(* IEC 61131-3 sources: 2026_Projet_YGO_ExcavatriceDragage/CODE/IO, 4 files *)

(* ---- GVL_IN.st ---- *)
(* ═══════════════════════════════════════════════════════════════
   🗂️ GVL_IN — Entrées machine CONDITIONNÉES (sortie de FB_InputsMachine)
   ───────────────────────────────────────────────────────────────
   📄 Doc : DOC/AF_Partie6_IO_Conditioning_v1.2.md §5
   🔴 ÉCRITURE : FB_InputsMachine SEULEMENT — ne jamais écrire ailleurs !
   ✅ LECTURE : tous les autres POUs (Safety, Winch, Chariot, Homing…)

   🔌 RÈGLE CÂBLAGE SÉCURITÉ (lire avant de modifier) :
   ─────────────────────────────────────────────────────
   Tous les capteurs de sécurité sont câblés en NORMALEMENT FERMÉ (NC) :
     ✅ REPOS / SAIN = TRUE (1) → circuit fermé, courant qui passe → tout va bien
     🔴 DÉFAUT / FIN DE COURSE = FALSE (0) → circuit ouvert (sécurité OU fil coupé)
   Avantage : une coupure de fil = une détection de défaut automatique !
   ═══════════════════════════════════════════════════════════════ *)

// === DECLARATION (à coller dans la partie déclaration du GVL GVL_IN) ===

VAR_GLOBAL

    // ─────────────────────────────────────────────────────────────────────
    // 🛑 SÉCURITÉS COMMUNES (NC — repos = TRUE, défaut/actionné = FALSE)
    // ─────────────────────────────────────────────────────────────────────

    EmergencyStopOk      : BOOL;
    // 🚨 Chaîne arrêt d'urgence (AU bouton champignon + filets de sécurité)
    //    TRUE  = chaîne AU FERMÉE → machine autorisée à bouger
    //    FALSE = chaîne AU COUPÉE (bouton appuyé OU câble coupé) → STOP immédiat

    TopPositionSensor    : BOOL;
    // 🔝 Capteur fin de course HAUT (NC monté en sécurité positive)
    //    TRUE  = capteur LIBRE → câble pas en butée haute, mouvement OK
    //    FALSE = capteur ACTIONNÉ (butée atteinte) → remontée interdite, homing déclenché

    SlackCableSwitch     : BOOL;
    // 🔗 Détecteur mou de câble (NC — repos = câble tendu)
    //    TRUE  = câble TENDU → OK pour descendre
    //    FALSE = câble MOU détecté → descente interdite, remontée autorisée uniquement
    //    ⚠️ Logique de commande : ForbidDescent := NOT SlackCableSwitch (voir FB_Safety_Winch)

    PhaseRotationOk      : BOOL;
    // ⚡ Relais contrôle rotation de phases électriques (NC)
    //    TRUE  = phases CORRECTES → moteurs autorisés à démarrer
    //    FALSE = phases inversées/absentes → SafeStop immédiat (moteurs tourneraient à l'envers !)

    // ─────────────────────────────────────────────────────────────────────
    // 🪝 TREUIL M1 — Retours contacteurs & sécurités (logique mixte NC/NO)
    // ─────────────────────────────────────────────────────────────────────

    M1ContactorFeedbackFwd : BOOL;
    // 📡 Retour contacteur MONTÉE M1 (NO miroir de la bobine)
    //    TRUE  = contacteur montée FERMÉ (bobine alimentée, courant de puissance qui passe)
    //    FALSE = contacteur ouvert (commande coupée ou contacteur collé si commande=TRUE)

    M1ContactorFeedbackRev : BOOL;
    // 📡 Retour contacteur DESCENTE M1 (NO miroir de la bobine)
    //    TRUE  = contacteur descente FERMÉ
    //    FALSE = contacteur ouvert

    M1ThermalFeedback      : BOOL;
    // 🌡️ Sonde thermique moteur M1 (NC — protection moteur contre surchauffe)
    //    TRUE  = température NORMALE → moteur autorisé
    //    FALSE = SURCHAUFFE ou fil coupé → SafeStop M1 immédiat

    M1BrakeFeedback        : BOOL;
    // 🔒 Retour contacteur frein électromagnétique M1 (NC — frein serré = sûr)
    //    TRUE  = frein SERRÉ (bobine coupée, ressort actif) → position sécurisée
    //    FALSE = frein DESSERRÉ (bobine alimentée, frein relâché pour mouvement)

    // ─────────────────────────────────────────────────────────────────────
    // 🪝 TREUIL M2 — Retours contacteurs & sécurités (même logique que M1)
    // ─────────────────────────────────────────────────────────────────────

    M2ContactorFeedbackFwd : BOOL;
    // 📡 Retour contacteur MONTÉE M2 — même logique que M1ContactorFeedbackFwd

    M2ContactorFeedbackRev : BOOL;
    // 📡 Retour contacteur DESCENTE M2 — même logique que M1ContactorFeedbackRev

    M2ThermalFeedback      : BOOL;
    // 🌡️ Sonde thermique moteur M2 — même logique que M1ThermalFeedback

    M2BrakeFeedback        : BOOL;
    // 🔒 Retour contacteur frein M2 — même logique que M1BrakeFeedback

    // ─────────────────────────────────────────────────────────────────────
    // ↔️ CHARIOT M3 — Capteurs de position (NO — actionné = position atteinte = TRUE)
    // ─────────────────────────────────────────────────────────────────────

    ChariotPosFosse1      : BOOL;
    // 📍 Capteur position FOSSE 1 (NO — position atteinte = TRUE)
    //    TRUE  = chariot EN POSITION fosse 1 (fin de course actionné physiquement)
    //    FALSE = chariot hors de la fosse 1

    ChariotPosFosse2      : BOOL;
    // 📍 Capteur position FOSSE 2 — même logique que ChariotPosFosse1

    ChariotPosMaintenance : BOOL;
    // 🔧 Capteur position MAINTENANCE — chariot en position de service
    //    TRUE  = position maintenance atteinte (pour interventions mécaniques)

    ChariotPosTremie      : BOOL;
    // 🗑️ Capteur position TRÉMIE (déversement) — chariot en position vidange
    //    TRUE  = position trémie atteinte → autorisation ouverture grappin

    M3BrakeFeedback       : BOOL;
    // 🔒 Retour contacteur frein chariot M3 — même logique que M1BrakeFeedback

END_VAR

(* ---- GVL_OUT.st ---- *)
(* ═══════════════════════════════════════════════════════════════
   🗂️ GVL_OUT — Commandes déjà rampées des FB métier (entrée de FB_OutputsMachine)
   ───────────────────────────────────────────────────────────────
   📄 Doc métier : DOC/AF_Partie6_IO_Conditioning_v1.2.md §5
   🔧 AJOUT (2026-07-03quindecies, demande utilisateur) : `PRG_MAIN` écrit ICI les
      commandes déjà rampées de `FB_Winch`/`FB_Chariot` par simples affectations
      (naturel en LD : 1 rung = 1 bobine), plutôt que de les passer en paramètres
      d'un appel de FB à 15 entrées (lourd à câbler en Ladder). `FB_OutputsMachine`
      lit ensuite ces variables directement en interne, appelée SANS paramètre.
   ⚠️ Écart assumé à Partie2 §0 ("quasi pas de GVL, sauf échange IHM") — même choix
      pragmatique que `GVL_IN`.
   🔴 Écrit UNIQUEMENT par `PRG_MAIN` (après `FB_Winch`/`FB_Chariot`), lu UNIQUEMENT
      par `FB_OutputsMachine`.
   ═══════════════════════════════════════════════════════════════ *)

// === DECLARATION (à coller dans la partie déclaration du GVL GVL_OUT) ===

VAR_GLOBAL
    // 🪝 WINCH M1
    M1RelayFwd        : BOOL;
    M1RelayRev        : BOOL;
    M1SpeedContactor1 : BOOL;
    M1SpeedContactor2 : BOOL;
    M1SpeedContactor3 : BOOL;
    M1SpeedContactor4 : BOOL;
    M1BrakeCmd        : BOOL;

    // 🪝 WINCH M2
    M2RelayFwd        : BOOL;
    M2RelayRev        : BOOL;
    M2SpeedContactor1 : BOOL;
    M2SpeedContactor2 : BOOL;
    M2SpeedContactor3 : BOOL;
    M2SpeedContactor4 : BOOL;
    M2BrakeCmd        : BOOL;

    // ↔️ CHARIOT M3 — seul BrakeCmd est réel
    ChariotBrakeCmd   : BOOL;
END_VAR

(* ---- FB_InputsMachine.st ---- *)
(* ═══════════════════════════════════════════════════════════════
   📥 FB_InputsMachine — Conditionnement ENTRÉES réelles de toute la machine (1 instance)
   ───────────────────────────────────────────────────────────────
   📄 Doc métier : DOC/AF_Partie6_IO_Conditioning_v1.2.md §5 (historique détaillé : AUDIT
      D52/D60/D61/D64)
   🧭 Interface RÉDUITE (Partie3 §1bis) : compose FB_Input (_COMMON) pour TOUTES les entrées
      TOR réelles (Commun/Winch M1/Winch M2/Chariot M3). Référence DIRECTEMENT les I/O réels
      globales en interne (pas de `*Raw`/`Invert*` câblés depuis `PRG_MAIN`) et écrit ses
      sorties DIRECTEMENT dans `GVL_IN.Xxx` (noms courts, sans suffixe) — appelé SANS
      PARAMÈTRE, rien à récupérer en retour. `InvertLogic`/`ChannelOk` de chaque sous-instance
      restent à leur défaut (FALSE/TRUE) — à FORCER DIRECTEMENT sur la sous-instance en vue
      CODESYS pour inverser NO/NC en mise en service, sans recompiler.
   ℹ️ Note utilisateur : prévu pour être implémenté en LANGAGE LD (Ladder) dans CODESYS pour
      faciliter la maintenance — code ci-dessous = référence ST. `FilterTime` : valeurs
      indicatives (`T#20MS`), à ajuster par voie selon le besoin réel (rebond capteur).
   🔴 NON CÂBLÉS ICI (pas de FB consommateur — FB_Grappin n'existe pas encore) :
      `ConveyorInfeedReady_DI`, `GridDwn_RQ`/`GridUp_RQ`, `HelmetClose_RQ`/`HelmetOpen_RQ`,
      `PosCasque_DI`, `PosGrille_DI`, `ThermHydraulique_DI`.
   ═══════════════════════════════════════════════════════════════ *)

// === DECLARATION (à coller dans la partie déclaration du POU FB_InputsMachine) ===

FUNCTION_BLOCK PUBLIC FB_InputsMachine
VAR
    // 🛑 Commun
    instEmergencyStopOk   : FB_Input;
    instSlackCableSwitch  : FB_Input;
    instTopPositionSensor : FB_Input;
    instCtrlPhaseRotation : FB_Input;   // 🆕 2026-07-03sexdecies — contrôle rotation phases élec.

    // 🪝 Winch M1
    instM1ContactorFwd : FB_Input;
    instM1ContactorRev : FB_Input;
    instM1Thermal      : FB_Input;
    instM1BrakeFeedback: FB_Input;

    // 🪝 Winch M2
    instM2ContactorFwd : FB_Input;
    instM2ContactorRev : FB_Input;
    instM2Thermal      : FB_Input;
    instM2BrakeFeedback: FB_Input;

    // ↔️ Chariot M3
    instChariotPosFosse1      : FB_Input;
    instChariotPosFosse2      : FB_Input;
    instChariotPosMaintenance : FB_Input;
    instChariotPosTremie      : FB_Input;
    instM3BrakeFeedback       : FB_Input;
END_VAR

// === IMPLEMENTATION (à coller dans le corps ST du POU FB_InputsMachine) ===

// 🛑 ─── COMMUN ────────────────────────────────────────────────────────────
// ⚠️ Bypass TEST banc (GVL_DEBUG) — TOUJOURS FALSE avant essai réel avec la chaîne AU câblée
instEmergencyStopOk(InputRaw := EmergencyStopOk_DI OR GVL_DEBUG.DBG_EmergencyStopOkBypass_TEST, FilterTime := T#20MS);
GVL_IN.EmergencyStopOk := instEmergencyStopOk.State;

// ⚠️ Bypass TEST banc (GVL_DEBUG, créé par l'utilisateur) — TOUJOURS FALSE avant essai réel
// avec le vrai capteur mou de câble câblé. Câblage sécurité : TRUE=OK (pas de mou) — le
// bypass force donc l'état OK, cohérent avec les autres bypass (OR sur le signal brut).
instSlackCableSwitch(InputRaw := M1_M2_SlackCableSwitch_DI OR GVL_DEBUG.DBG_SlackCableSwitch_TEST, FilterTime := T#20MS);
GVL_IN.SlackCableSwitch := instSlackCableSwitch.State;

// ⚠️ Bypass TEST banc (GVL_DEBUG) — TOUJOURS FALSE avant essai réel avec le capteur câblé
instTopPositionSensor(InputRaw := M1_M2_TopPositionSensor_DI OR GVL_DEBUG.DBG_TopPositionSensorBypass_TEST, FilterTime := T#20MS);
GVL_IN.TopPositionSensor := instTopPositionSensor.State;

// 🆕 Contrôle rotation phases électriques (2026-07-03sexdecies) — TRUE = rotation correcte.
// Câblé dans FB_Safety_Winch/FB_Safety_Chariot (D71), pas directement sur EmergencyStopOk.
// ⚠️ Bypass TEST banc (GVL_DEBUG, créé par l'utilisateur) — TOUJOURS FALSE avant essai réel
// avec le vrai contrôle de rotation câblé.
instCtrlPhaseRotation(InputRaw := CtrlPhaseRotation_DI OR GVL_DEBUG.DBG_CtrlPhaseRotation_Bypass_TEST, FilterTime := T#20MS);
GVL_IN.PhaseRotationOk := instCtrlPhaseRotation.State;

// 🪝 ─── WINCH M1 ──────────────────────────────────────────────────────────
instM1ContactorFwd(InputRaw := M1_ContactorFeedbackFwd_DI, FilterTime := T#20MS);
GVL_IN.M1ContactorFeedbackFwd := instM1ContactorFwd.State;

instM1ContactorRev(InputRaw := M1_ContactorFeedbackRev_DI, FilterTime := T#20MS);
GVL_IN.M1ContactorFeedbackRev := instM1ContactorRev.State;

instM1Thermal(InputRaw := M1_ThermalFeedback_DI, FilterTime := T#20MS);
GVL_IN.M1ThermalFeedback := instM1Thermal.State;

// 🆕 Retour frein M1 RÉEL (était miroir logiciel GVL_Winch_M1_Stub)
instM1BrakeFeedback(InputRaw := M1_BrakeContactorFeedback_DI, FilterTime := T#20MS);
GVL_IN.M1BrakeFeedback := instM1BrakeFeedback.State;

// 🪝 ─── WINCH M2 ──────────────────────────────────────────────────────────
instM2ContactorFwd(InputRaw := M2_ContactorFeedbackFwd_DI, FilterTime := T#20MS);
GVL_IN.M2ContactorFeedbackFwd := instM2ContactorFwd.State;

instM2ContactorRev(InputRaw := M2_ContactorFeedbackRev_DI, FilterTime := T#20MS);
GVL_IN.M2ContactorFeedbackRev := instM2ContactorRev.State;

instM2Thermal(InputRaw := M2_ThermalFeedback_DI, FilterTime := T#20MS);
GVL_IN.M2ThermalFeedback := instM2Thermal.State;

// 🆕 Retour frein M2 RÉEL (était miroir logiciel GVL_Winch_M2_Stub)
instM2BrakeFeedback(InputRaw := M2_BrakeContactorFeedback_DI, FilterTime := T#20MS);
GVL_IN.M2BrakeFeedback := instM2BrakeFeedback.State;

// ↔️ ─── CHARIOT M3 — 4 capteurs position réels ───────────────────────────
instChariotPosFosse1(InputRaw := PosFosse1_DI, FilterTime := T#20MS);
GVL_IN.ChariotPosFosse1 := instChariotPosFosse1.State;

instChariotPosFosse2(InputRaw := PosFosse2_DI, FilterTime := T#20MS);
GVL_IN.ChariotPosFosse2 := instChariotPosFosse2.State;

instChariotPosMaintenance(InputRaw := PosMaintenance_DI, FilterTime := T#20MS);
GVL_IN.ChariotPosMaintenance := instChariotPosMaintenance.State;

instChariotPosTremie(InputRaw := PosTremie_DI, FilterTime := T#20MS);
GVL_IN.ChariotPosTremie := instChariotPosTremie.State;

// 🆕 Retour frein M3 RÉEL (était miroir logiciel GVL_Chariot_M3_Stub)
instM3BrakeFeedback(InputRaw := M3_BrakeContactorFeedback_DI, FilterTime := T#20MS);
GVL_IN.M3BrakeFeedback := instM3BrakeFeedback.State;

(* ---- PRG_0_Inputs.st ---- *)
(* ═══════════════════════════════════════════════════════════════
   📥 PRG_0_Inputs — Acquisition et conditionnement des ENTRÉES (PROGRAMME)
   ───────────────────────────────────────────────────────────────
   📄 Doc : DOC/AF_Partie6_IO_Conditioning_v1.2.md §5
   ⚙️ Exécuté par la tâche PLC (Task Manager) en position 0.
   ✅ Expose ses sorties en VAR_OUTPUT (lecture seule pour le reste du code).
   ═══════════════════════════════════════════════════════════════ *)

PROGRAM PRG_0_Inputs
VAR_OUTPUT
    // ── 🛑 SÉCURITÉS COMMUNES (NC — repos=TRUE sain, FALSE=défaut/fil coupé) ──────────────
    EmergencyStopOk      : BOOL;   // 🚨 Chaîne AU : TRUE=fermée/armée ✅ | FALSE=AU appuyé ou fil coupé 🔴
    TopPositionSensor    : BOOL;   // 🔝 Fin de course HAUT (NC) : TRUE=libre ✅ | FALSE=butée atteinte 🔴→ForbidAscent
    SlackCableSwitch     : BOOL;   // 🔗 Mou câble sur tambour M2 (NC) : TRUE=câble tendu ✅ | FALSE=mou détecté 🔴→ForbidDescent
    PhaseRotationOk      : BOOL;   // ⚡ Rotation phases élec. (NC) : TRUE=phases OK ✅ | FALSE=inversées/absentes 🔴→SafeStop

    // ── 🪝 TREUIL M1 (contacteurs=NO miroir bobine ; thermique/frein=NC) ────────────────
    M1ContactorFeedbackFwd : BOOL; // 📡 Retour contacteur MONTÉE M1 (NO) : TRUE=contacteur fermé | FALSE=ouvert
    M1ContactorFeedbackRev : BOOL; // 📡 Retour contacteur DESCENTE M1 (NO) : TRUE=contacteur fermé | FALSE=ouvert
    M1ThermalFeedback      : BOOL; // 🌡️ Thermique moteur M1 (NC) : TRUE=temp OK ✅ | FALSE=surchauffe ou coupure 🔴
    M1BrakeFeedback        : BOOL; // 🔒 Retour frein M1 (NC) : TRUE=frein serré repos ✅ | FALSE=desserré/coupure 🔴

    // ── 🪝 TREUIL M2 (même logique que M1) ──────────────────────────────────────────────
    M2ContactorFeedbackFwd : BOOL; // 📡 Retour contacteur MONTÉE M2 (NO) : TRUE=fermé | FALSE=ouvert
    M2ContactorFeedbackRev : BOOL; // 📡 Retour contacteur DESCENTE M2 (NO) : TRUE=fermé | FALSE=ouvert
    M2ThermalFeedback      : BOOL; // 🌡️ Thermique moteur M2 (NC) : TRUE=temp OK ✅ | FALSE=surchauffe ou coupure 🔴
    M2BrakeFeedback        : BOOL; // 🔒 Retour frein M2 (NC) : TRUE=serré repos ✅ | FALSE=desserré/coupure 🔴

    // ── ↔️ CHARIOT M3 (capteurs position=NO — position atteinte=TRUE) ────────────────────
    ChariotPosFosse1      : BOOL;  // 📍 Position fosse 1 (NO) : TRUE=chariot en fosse 1 ✅ | FALSE=absent
    ChariotPosFosse2      : BOOL;  // 📍 Position fosse 2 (NO) : TRUE=chariot en fosse 2 ✅ | FALSE=absent
    ChariotPosMaintenance : BOOL;  // 🔧 Position maintenance (NO) : TRUE=en position service ✅ | FALSE=absent
    ChariotPosTremie      : BOOL;  // 🗑️ Position trémie vidange (NO) : TRUE=en position trémie ✅ | FALSE=absent
    M3BrakeFeedback       : BOOL;  // 🔒 Retour frein chariot M3 (NC) : TRUE=serré repos ✅ | FALSE=desserré 🔴
END_VAR
VAR
    // Instances de filtrage
    instEmergencyStopOk   : FB_Input;
    instSlackCableSwitch  : FB_Input;
    instTopPositionSensor : FB_Input;
    instCtrlPhaseRotation : FB_Input;

    instM1ContactorFwd : FB_Input;
    instM1ContactorRev : FB_Input;
    instM1Thermal      : FB_Input;
    instM1BrakeFeedback: FB_Input;

    instM2ContactorFwd : FB_Input;
    instM2ContactorRev : FB_Input;
    instM2Thermal      : FB_Input;
    instM2BrakeFeedback: FB_Input;

    instChariotPosFosse1      : FB_Input;
    instChariotPosFosse2      : FB_Input;
    instChariotPosMaintenance : FB_Input;
    instChariotPosTremie      : FB_Input;
    instM3BrakeFeedback       : FB_Input;
END_VAR

// === IMPLEMENTATION (corps du PROGRAM PRG_0_Inputs) ===

// 🛑 ─── COMMUN ────────────────────────────────────────────────────────────
instEmergencyStopOk(InputRaw := EmergencyStopOk_DI OR GVL_DEBUG.DBG_EmergencyStopOkBypass_TEST, FilterTime := T#20MS);
EmergencyStopOk := instEmergencyStopOk.State;

instSlackCableSwitch(InputRaw := M1_M2_SlackCableSwitch_DI OR GVL_DEBUG.DBG_SlackCableSwitch_TEST, FilterTime := T#20MS);
SlackCableSwitch := instSlackCableSwitch.State;

instTopPositionSensor(InputRaw := M1_M2_TopPositionSensor_DI OR GVL_DEBUG.DBG_TopPositionSensorBypass_TEST, FilterTime := T#20MS);
TopPositionSensor := instTopPositionSensor.State;

instCtrlPhaseRotation(InputRaw := CtrlPhaseRotation_DI OR GVL_DEBUG.DBG_CtrlPhaseRotation_Bypass_TEST, FilterTime := T#20MS);
PhaseRotationOk := instCtrlPhaseRotation.State;

// 🪝 ─── WINCH M1 ──────────────────────────────────────────────────────────
instM1ContactorFwd(InputRaw := M1_ContactorFeedbackFwd_DI, FilterTime := T#20MS);
M1ContactorFeedbackFwd := instM1ContactorFwd.State;

instM1ContactorRev(InputRaw := M1_ContactorFeedbackRev_DI, FilterTime := T#20MS);
M1ContactorFeedbackRev := instM1ContactorRev.State;

instM1Thermal(InputRaw := M1_ThermalFeedback_DI OR GVL_DEBUG.DBG_ContactorFeedbackBypass_TEST, FilterTime := T#20MS);
M1ThermalFeedback := instM1Thermal.State;

instM1BrakeFeedback(InputRaw := M1_BrakeContactorFeedback_DI, FilterTime := T#20MS);
M1BrakeFeedback := instM1BrakeFeedback.State;

// 🪝 ─── WINCH M2 ──────────────────────────────────────────────────────────
instM2ContactorFwd(InputRaw := M2_ContactorFeedbackFwd_DI, FilterTime := T#20MS);
M2ContactorFeedbackFwd := instM2ContactorFwd.State;

instM2ContactorRev(InputRaw := M2_ContactorFeedbackRev_DI, FilterTime := T#20MS);
M2ContactorFeedbackRev := instM2ContactorRev.State;

instM2Thermal(InputRaw := M2_ThermalFeedback_DI OR GVL_DEBUG.DBG_ContactorFeedbackBypass_TEST, FilterTime := T#20MS);
M2ThermalFeedback := instM2Thermal.State;

instM2BrakeFeedback(InputRaw := M2_BrakeContactorFeedback_DI, FilterTime := T#20MS);
M2BrakeFeedback := instM2BrakeFeedback.State;

// ↔️ ─── CHARIOT M3 ────────────────────────────────────────────────────────
instChariotPosFosse1(InputRaw := PosFosse1_DI, FilterTime := T#20MS);
ChariotPosFosse1 := instChariotPosFosse1.State;

instChariotPosFosse2(InputRaw := PosFosse2_DI, FilterTime := T#20MS);
ChariotPosFosse2 := instChariotPosFosse2.State;

instChariotPosMaintenance(InputRaw := PosMaintenance_DI, FilterTime := T#20MS);
ChariotPosMaintenance := instChariotPosMaintenance.State;

instChariotPosTremie(InputRaw := PosTremie_DI, FilterTime := T#20MS);
ChariotPosTremie := instChariotPosTremie.State;

instM3BrakeFeedback(InputRaw := M3_BrakeContactorFeedback_DI, FilterTime := T#20MS);
M3BrakeFeedback := instM3BrakeFeedback.State;
